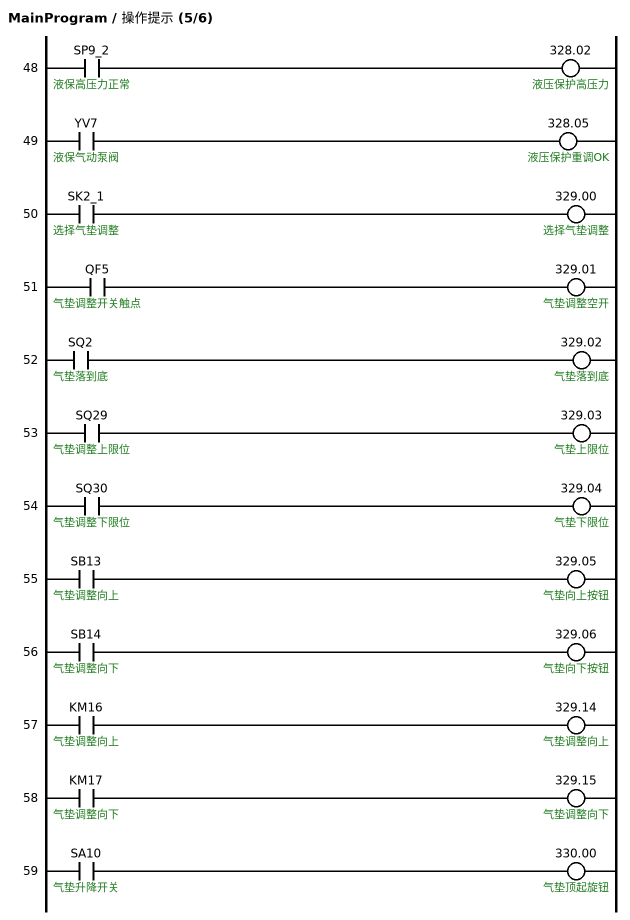
; [picture p48: MainProgram / 操作提示, rungs 48-59]
; rung 48
LD SP9_2  ; 液保高压力正常
OUT 328.02  ; 液压保护高压力
; rung 49
LD YV7  ; 液保气动泵阀
OUT 328.05  ; 液压保护重调OK
; rung 50
LD SK2_1  ; 选择气垫调整
OUT 329.00  ; 选择气垫调整
; rung 51
LD QF5  ; 气垫调整开关触点
OUT 329.01  ; 气垫调整空开
; rung 52
LD SQ2  ; 气垫落到底
OUT 329.02  ; 气垫落到底
; rung 53
LD SQ29  ; 气垫调整上限位
OUT 329.03  ; 气垫上限位
; rung 54
LD SQ30  ; 气垫调整下限位
OUT 329.04  ; 气垫下限位
; rung 55
LD SB13  ; 气垫调整向上
OUT 329.05  ; 气垫向上按钮
; rung 56
LD SB14  ; 气垫调整向下
OUT 329.06  ; 气垫向下按钮
; rung 57
LD KM16  ; 气垫调整向上
OUT 329.14  ; 气垫调整向上
; rung 58
LD KM17  ; 气垫调整向下
OUT 329.15  ; 气垫调整向下
; rung 59
LD SA10  ; 气垫升降开关
OUT 330.00  ; 气垫顶起旋钮

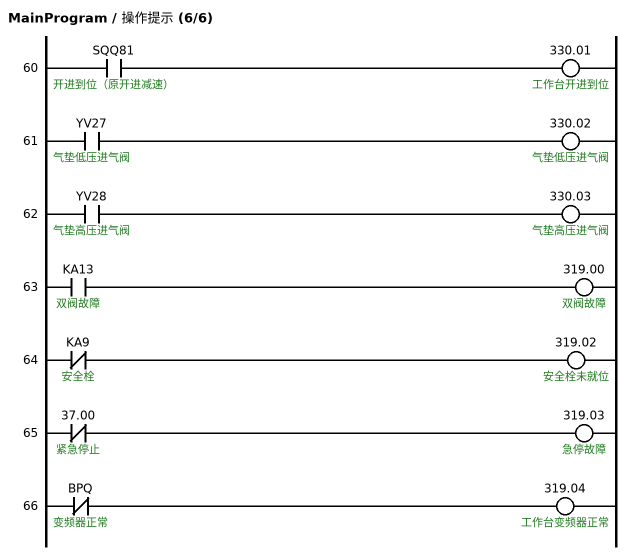
; rung 60
LD SQQ81  ; 开进到位（原开进减速）
OUT 330.01  ; 工作台开进到位
; rung 61
LD YV27  ; 气垫低压进气阀
OUT 330.02  ; 气垫低压进气阀
; rung 62
LD YV28  ; 气垫高压进气阀
OUT 330.03  ; 气垫高压进气阀
; rung 63
LD KA13  ; 双阀故障
OUT 319.00  ; 双阀故障
; rung 64
LDNOT KA9  ; 安全栓
OUT 319.02  ; 安全栓未就位
; rung 65
LDNOT 37.00  ; 紧急停止
OUT 319.03  ; 急停故障
; rung 66
LDNOT BPQ  ; 变频器正常
OUT 319.04  ; 工作台变频器正常

### Section 模具加紧

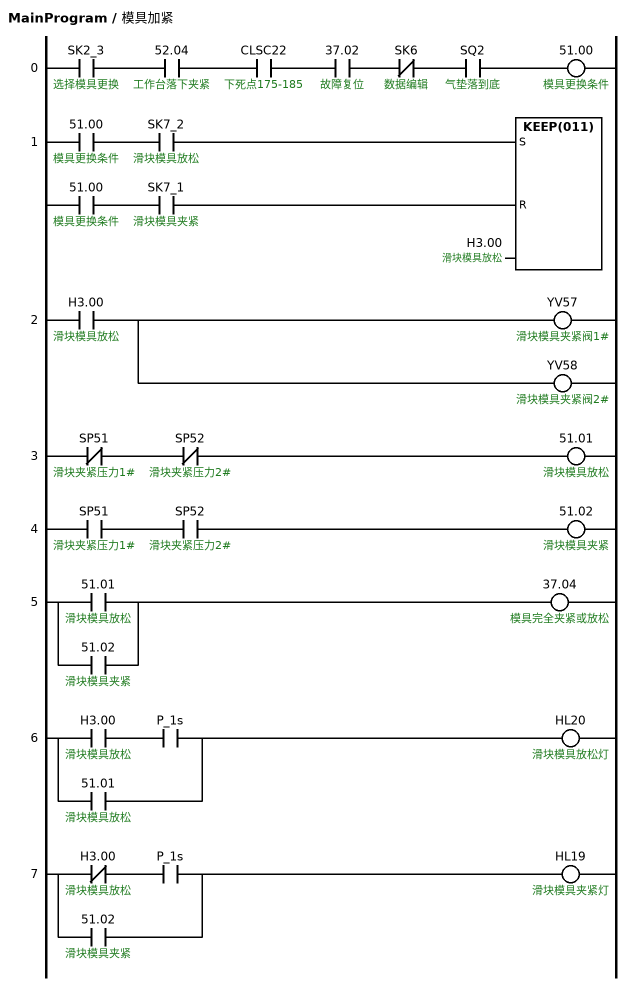
; rung 0
LD SK2_3  ; 选择模具更换
AND 52.04  ; 工作台落下夹紧
AND CLSC22  ; 下死点175-185
AND 37.02  ; 故障复位
ANDNOT SK6  ; 数据编辑
AND SQ2  ; 气垫落到底
OUT 51.00  ; 模具更换条件
; rung 1
LD 51.00  ; 模具更换条件
AND SK7_2  ; 滑块模具放松
LD 51.00  ; 模具更换条件
AND SK7_1  ; 滑块模具夹紧
KEEP(011) H3.00  ; 滑块模具放松
; rung 2
LD H3.00  ; 滑块模具放松
OUT YV57  ; 滑块模具夹紧阀1#
OUT YV58  ; 滑块模具夹紧阀2#
; rung 3
LDNOT SP51  ; 滑块夹紧压力1#
ANDNOT SP52  ; 滑块夹紧压力2#
OUT 51.01  ; 滑块模具放松
; rung 4
LD SP51  ; 滑块夹紧压力1#
AND SP52  ; 滑块夹紧压力2#
OUT 51.02  ; 滑块模具夹紧
; rung 5
LD 51.01  ; 滑块模具放松
OR 51.02  ; 滑块模具夹紧
OUT 37.04  ; 模具完全夹紧或放松
; rung 6
LD H3.00  ; 滑块模具放松
AND P_1s
OR 51.01  ; 滑块模具放松
OUT HL20  ; 滑块模具放松灯
; rung 7
LDNOT H3.00  ; 滑块模具放松
AND P_1s
OR 51.02  ; 滑块模具夹紧
OUT HL19  ; 滑块模具夹紧灯

### Section 结束
; rung 0
END(001)